# EPICS autosave request: app/Db/CARBIDE.req
$$LOOP(REG)
$$IF(DIR,RW)
$$IF(NOARCH)
$$ELSE(NOARCH)
$(BASE):$$NAME
$$ENDIF(NOARCH)
$$ENDIF(DIR)
$$ENDLOOP(REG)
